Staubli VAL3: onF6Event.pgx

program onF6Event()
  local num l_nSize
begin
  // look if the bButton is enable
  if bButton[5]
   //
    if cycleStatus:bSimulation and cycleStatus:bPause and esStatus()!=2
      call OnEvent:resumeCycle()
    endIf
  endIf
end
